// TIA Portal V20 export
// export: Created 2025-12-01T14:56:13.5985525Z, ExportSetting None, DisplayName Totally Integrated Automation Portal, DisplayVersion V20 Update 3, DisplayName TIA Portal Openness, DisplayVersion V20 Update 3, DisplayName TIA Portal Version Control Interface, DisplayVersion V20 Update 3, DisplayName STEP 7 Professional, DisplayVersion V20 Update 3, DisplayName STEP 7 Safety, DisplayVersion V20 Update 2, DisplayName WinCC Basic/Comfort/Advanced, DisplayVersion V20 Update 3, DisplayName WinCC Professional, DisplayVersion V20 Update 3, DisplayName WinCC Unified, DisplayVersion V20 Update 3
TYPE "UDT_EventosMemoria"
   STRUCT
      Tipo : UInt;   // Tipo de Memoria a Leer
      Numero : UInt;   // Numero de la Memmoria a Leer
      Offset : UInt;   // Offset dentro de la Memoria a partir de donde debe Leerse
      Longitud : UInt;   // Longitud de memoria que debe Leerse
   END_STRUCT;
END_TYPE
